TYPE "UDT300_EM_Heating"
VERSION : 2.0
STRUCT
    HW_Freeze_Stat_DI : Bool;     // Digital Input: Freeze-stat on hot water coil (`True` = Fault).
    HW_Valve_Fdbk_AI : Real;      // Analog Input: Hot water valve position feedback (0.0 - 100.0 %).
    HW_Valve_Cmd_AO : Real;       // Analog Output: Hot water valve position command (0.0 - 100.0 %).
    HW_Freeze_Alm : Bool;         // Alarm: Hot water coil freeze-stat tripped.
END_STRUCT
END_TYPE